// LS Electric XG5000 project: 주차설비
// PLC LSPLC

PROGRAM NewProgram (task: 스캔 프로그램)

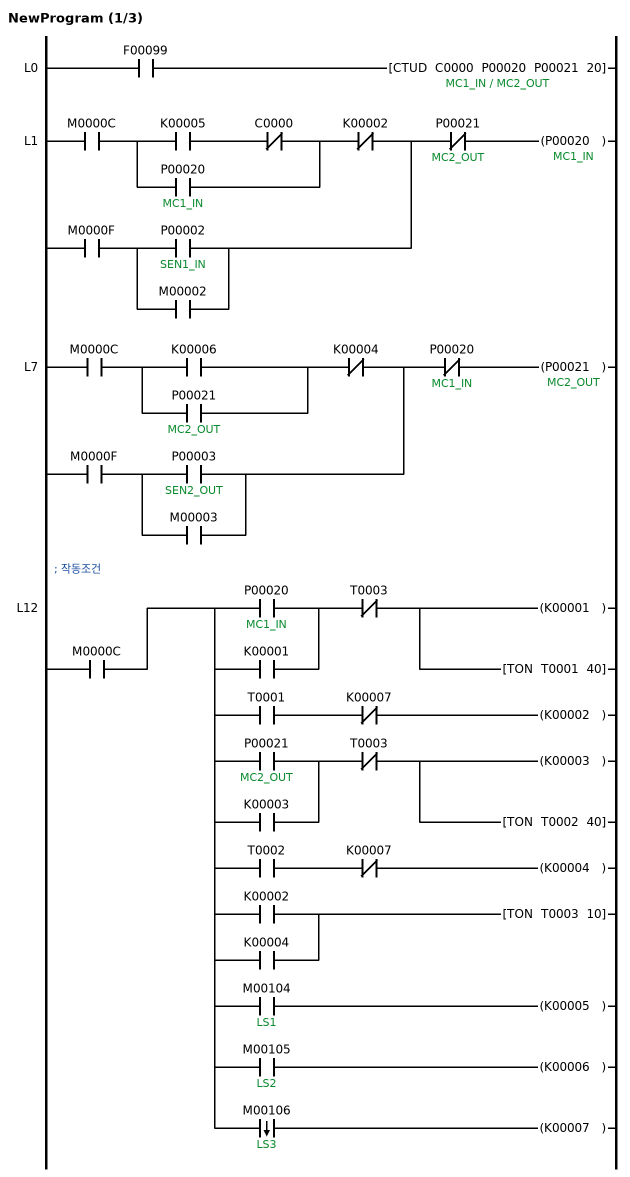
; L0
LOAD      F00099
CTUD      C0000 P00020 P00021 20	// MC1_IN / MC2_OUT
; L1
LOAD      M0000C
LOAD      K00005
AND NOT   C0000
OR        P00020	// MC1_IN
AND LOAD
AND NOT   K00002
LOAD      M0000F
LOAD      P00002	// SEN1_IN
OR        M00002
AND LOAD
OR LOAD
AND NOT   P00021	// MC2_OUT
OUT       P00020	// MC1_IN
; L7
LOAD      M0000C
LOAD      K00006
OR        P00021	// MC2_OUT
AND LOAD
AND NOT   K00004
LOAD      M0000F
LOAD      P00003	// SEN2_OUT
OR        M00003
AND LOAD
OR LOAD
AND NOT   P00020	// MC1_IN
OUT       P00021	// MC2_OUT
// 작동조건
; L12
LOAD      M0000C
MPUSH
LOAD      P00020	// MC1_IN
OR        K00001
AND LOAD
AND NOT   T0003
OUT       K00001
TON       T0001 40
MLOAD
AND       T0001
AND NOT   K00007
OUT       K00002
MLOAD
LOAD      P00021	// MC2_OUT
OR        K00003
AND LOAD
AND NOT   T0003
OUT       K00003
TON       T0002 40
MLOAD
AND       T0002
AND NOT   K00007
OUT       K00004
MLOAD
LOAD      K00002
OR        K00004
AND LOAD
TON       T0003 10
MLOAD
AND       M00104	// LS1
OUT       K00005
MLOAD
AND       M00105	// LS2
OUT       K00006
MPOP
ANDN      M00106	// LS3
OUT       K00007

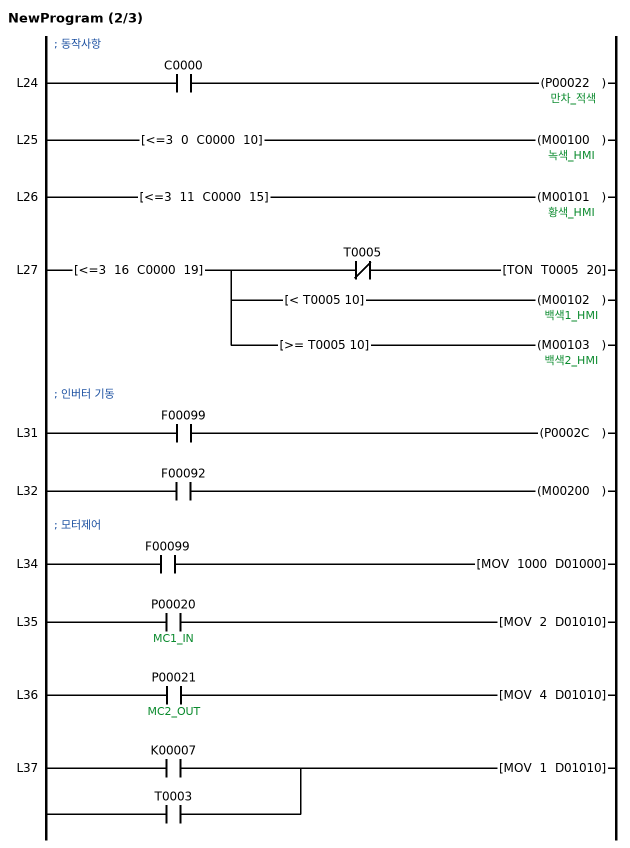
// 동작사항
; L24
LOAD      C0000
OUT       P00022	// 만차_적색
; L25
LOAD<=3   0 C0000 10
OUT       M00100	// 녹색_HMI
; L26
LOAD<=3   11 C0000 15
OUT       M00101	// 황색_HMI
; L27
LOAD<=3   16 C0000 19
MPUSH
AND NOT   T0005
TON       T0005 20
MLOAD
AND<      T0005 10
OUT       M00102	// 백색1_HMI
MPOP
AND>=     T0005 10
OUT       M00103	// 백색2_HMI
// 인버터 기동
; L31
LOAD      F00099
OUT       P0002C
; L32
LOAD      F00092
OUT       M00200
// 모터제어
; L34
LOAD      F00099
MOV       1000 D01000
; L35
LOAD      P00020	// MC1_IN
MOV       2 D01010
; L36
LOAD      P00021	// MC2_OUT
MOV       4 D01010
; L37
LOAD      K00007
OR        T0003
MOV       1 D01010

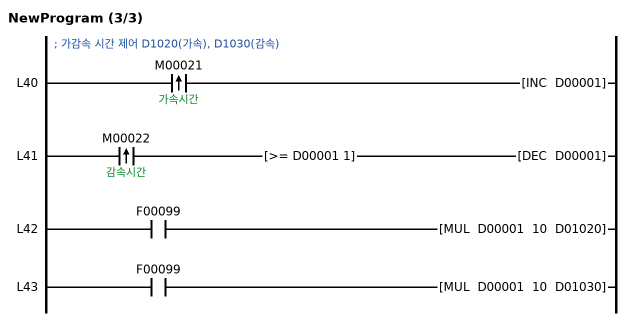
// 가감속 시간 제어 D1020(가속), D1030(감속)
; L40
LOADP     M00021	// 가속시간
INC       D00001
; L41
LOADP     M00022	// 감속시간
AND>=     D00001 1
DEC       D00001
; L42
LOAD      F00099
MUL       D00001 10 D01020
; L43
LOAD      F00099
MUL       D00001 10 D01030

VARIABLES AND COMMENTS (devices not used above)
P0000B	BIT	수동_자동
P00000	BIT	입차_IN
P00001	BIT	출차_OUT